{attribute 'GeneratedUsingTerminal: KL6211-0024'}
{attribute addProperty BoxType "KL6211-0024"}
{attribute addProperty Id "Channel_1AT %Q*Channel_A42BCA5C0"}
{attribute addProperty CRC "722560380"}
{attribute addProperty Size "0"}
TYPE KL_2B11657C :
STRUCT
	{attribute addProperty Name "Channel_1"}
	Channel_1 : Channel_A42BCA5C;
END_STRUCT
END_TYPE

(* stored: Version 1.2.0.0, ProductVersion 3.1.4024.9
   DUT KL_2B11657C: Id {684638e6-ee1f-45e3-99ee-15669c9f15be} *)
